// TwinCAT 3 PLC project AutoTune_PLC
// ProgramVersion: 3.1.4026.17
// libraries:
//   Tc2_MC2, * (Beckhoff Automation GmbH)
//   Tc2_Standard, * (Beckhoff Automation GmbH)
//   Tc2_System, * (Beckhoff Automation GmbH)
//   Tc3_Module, * (Beckhoff Automation GmbH)
//   VisuDialogs, * (System)
//   VisuSymbols,newest,System
// project tree:
//   / GlobalTextList.TcGTLO (not stored), PlcTask.TcTTO (not stored), Visualization Manager.TcVMO (not stored)
//   GVLs/ GVLSafeIO.TcGVL (not stored), GVLStdIO.TcGVL (not stored)
//   POUs/ FB_Blinker.TcPOU (not stored), MAIN.TcPOU
//   VISUs/ Visualization.TcVIS (not stored)
// real-time tasks:
//   TASK PlcTask: cycle T#10ms, priority 40, ADS port 350
// motion (NC):
//   TASK NC-Task 1 SAF: cycle T#2ms, priority 4, ADS port 501
//   TASK NC-Task 1 SVB: cycle T#10ms, priority 8, ADS port 511
//   AXIS Axis 1 (id 1)
//     General: UnitName=°
//     Dynamic: Acceleration=15000, Deceleration=15000, Jerk=69686.919
//     Velo: RefSearch=154.85982, RefSync=154.85982, SlowManual=774.2991, FastManual=4645.7946, Fast=15485.982, Maximum=15485.982
//     OtherSettings: AllowMotionCmdToSlave=true
//     encoder EncType=19
//       EncPara: ScaleFactorNumerator=360, ScaleFactorDenominator=1048576, MaxCount=#xffffffff
//     drive DrvType=16
//       DrvPara: MaxCount=#xffffffff, DriveControlDWord=#x00020100
//         Analog: VeloReferenz=17034.5802, VeloScale=71.5255737304688, TorqueSetpointScale=10, ScaleFactorActTorque=0.1
//         TimeComp: TaskDelayCycles=1
//     controller CtrType=1
//       CtrPara: PriorControlFactor=1
//         Observer: BandWidth=20
//   AXIS Axis 2 (id 2)
//     OtherSettings: AllowMotionCmdToSlave=true
//     encoder EncType=19
//       EncPara: MaxCount=#xffffffff
//     drive DrvType=16
//       DrvPara: MaxCount=#xffffffff, DriveControlDWord=#x00020100
//         Analog: TorqueSetpointScale=10, ScaleFactorActTorque=0.1
//         TimeComp: TaskDelayCycles=1
//     controller CtrType=1
//       CtrPara: PriorControlFactor=1
//         Observer: BandWidth=20
// I/O:
//   DEVICE Device 1 (EtherCAT), AmsNetId 5.143.164.192.2.1
//     Term 1 (EK1200) [EK1200-5000 EtherCAT Power supply (2A E-Bus)]
//       Term 2 (EL3214-0090) [EL3214-0090 4Ch. Ana. Input PT100 (RTD), TwinSAFE SC]
//       Term 3 (EL1904) [EL1904, 4 Ch. Safety Input 24V, TwinSAFE]
//         modules: Module 1 (FSOES)
//       Term 4 (EL2008) [EL2008 8Ch. Dig. Output 24V, 0.5A]
//       Term 5 (EL9011) [EL9011 End Terminal]
//   DEVICE Device 4 (EtherCAT), AmsNetId 5.143.164.192.5.1
//     Term 6 (AX8620-0000-0105) [AX8620-0000-0105]
//       Drive 7 (AX8206-0200-0106) [AX8206-0200-0106 (2Ch. 6A servo axis, safe-motion)]
//         modules: Device, Device, Device, Device, Device, Device, Device, Device, Device, Device, Device (Safety), Device, Device, Device, Device, Device, Device, Device, Device, Device, Device, Device, Device, Device, Device, Device, Device, Device, Device, Device, Device, Ch A, Ch A, Ch A, Ch A, Ch A, Ch A, Ch A, Ch A, Ch A, Ch A, Ch A, Ch A, Ch A, Ch A, Ch A, Ch A, Ch A, Ch A, Ch A, Ch A, Ch A, Ch A, Ch A, Ch A, Ch A, Ch A, Ch A, Ch A, Ch A, Ch A, Ch A, Ch B, Ch B, Ch B, Ch B, Ch B, Ch B, Ch B, Ch B, Ch B, Ch B, Ch B, Ch B, Ch B, Ch B, Ch B, Ch B, Ch B, Ch B, Ch B, Ch B, Ch B, Ch B, Ch B, Ch B, Ch B, Ch B
//         startup 12992:1 := 414D383034322D784A7830 // Ch A Motor parameters / Configured motor type
//         startup 24768:0 := FEFF // Ch A Interpolation sub mode select
//         startup 13000:5 := 0200 // Ch A Motor thermal model / Reaction
//         startup 13000:6 := 0000C841 // Ch A Motor thermal model / Partial fraction factor
//         startup 12992:12 := 0000FA45 // Ch A Motor parameters / Motor rated speed
//         startup 12992:13 := E6AE4540 // Ch A Motor parameters / Motor rated torque
//         startup 24694:0 := 03100000 // Ch A Motor standstill torque
//         startup 24800:0 := D007 // Ch A Positive torque/force limit value
//         startup 24801:0 := D007 // Ch A Negative torque/force limit value
//         startup 12288:6 := 4158383230362D303230302D30303030 // Ch A AxisMain parameters / Configured drive type
//         startup 12867:1 := CDCCDC40 // Ch A TorqueCtrl parameters / Configured channel rated current
//         startup 12867:2 := 0000A041 // Ch A TorqueCtrl parameters / Configured channel peak current
//         startup 12867:7 := 77BE1F40 // Ch A TorqueCtrl parameters / Iuvw max sum
//         startup 24672:0 := 08 // Ch A Modes of operation
//         startup 13023:0 := 0000 // Ch A Motor control mode
//         startup 12864:1 := 84C3B441 // Ch A TorqueCtrl parameters mappable / Torque control proportional gain q
//         startup 12864:2 := 8A0E7C39 // Ch A TorqueCtrl parameters mappable / Torque control integral action time q
//         startup 12608:1 := 9513BE3D // Ch A VeloCtrl parameters mappable / Velocity control proportional gain
//         startup 12608:2 := 6F12033C // Ch A VeloCtrl parameters mappable / Velocity control integral action time
//         startup 12608:3 := 00980546 // Ch A VeloCtrl parameters mappable / Bipolar velocity limit value
//         startup 12992:15 := 0100 // Ch A Motor parameters / Motor temperature sensor connection
//         startup 12611:4 := 0400 // Ch A VeloCtrl observer / Observer type
//         startup 24672:0 := 08 // Ch A Modes of operation
//         startup 12296:2 := 00 // Ch A AxisMain parameters encoder direction / Primary encoder direction
//   DEVICE Device 2 (EtherCAT Automation Protocol) (disabled), AmsNetId 5.143.164.192.3.1
//   DEVICE Device 3 (COM Port) (disabled)
//   DEVICE Device 7 (COM Port) (disabled)
// variable links:
//   Device 1 (EtherCAT) <-> Device 4 (EtherCAT)/Term 6 (AX8620-0000-0105)/Drive 7 (AX8206-0200-0106)
//     Term 1 (EK1200)/Term 3 (EL1904)/Module 1 (FSOES)/RxPDO/FSOE <-> Device (Safety)/FSoE Master Connection 1 Master Message/Message_3
//     Term 1 (EK1200)/Term 3 (EL1904)/Module 1 (FSOES)/TxPDO/FSOE <-> Device (Safety)/FSoE Master Connection 1 Slave Message/Message_3
//   Device 4 (EtherCAT) <-> Device 4 (EtherCAT)/Term 6 (AX8620-0000-0105)
//     Term 6 (AX8620-0000-0105)/Drive 7 (AX8206-0200-0106)/Device/DeviceMain Outputs/Power supply controlword <-> PSM Controlword for axis/Controlword for axis
//   NC-Task 1 SAF/Axes/Axis 1 <-> Device 4 (EtherCAT)/Term 6 (AX8620-0000-0105)/Drive 7 (AX8206-0200-0106)
//     Drive/Inputs/In/nDataIn1 <-> Ch A/Ch A PositionControl Inputs/Ch A Following error actual value
//     Drive/Inputs/In/nDataIn3[0] <-> Ch A/Ch A TorqueControl Inputs/Ch A Torque/force actual value
//     Drive/Inputs/In/nDcOutputTime <-> InfoData/DcOutputShift
//     Drive/Inputs/In/nState1 <-> Ch A/Ch A AxisMain Inputs/Ch A Statusword
//     Drive/Inputs/In/nState2 <-> Ch A/Ch A AxisMain Inputs/Ch A Statusword @bit 8
//     Drive/Inputs/In/nState4 @bit 1 <-> WcState/InputToggle0
//     Drive/Inputs/In/nState4 <-> WcState/WcState0
//     Drive/Outputs/Out/nCtrl1 <-> Ch A/Ch A AxisMain Outputs/Ch A Controlword
//     Drive/Outputs/Out/nCtrl2 <-> Ch A/Ch A AxisMain Outputs/Ch A Controlword @bit 8
//     Drive/Outputs/Out/nDataOut1 <-> Ch A/Ch A Interpolator Outputs/Ch A Target position
//     Drive/Outputs/Out/nDataOut2 <-> Ch A/Ch A Interpolator Outputs/Ch A Target velocity
//     Enc/Inputs/In/nDataIn1 <-> Ch A/Ch A AxisMain Inputs/Ch A Position actual value
//     Enc/Inputs/In/nDcInputTime <-> InfoData/DcInputShift
//     Enc/Inputs/In/nState2 @bit 5 <-> Ch A/Ch A AxisMain Inputs/Position actual value invalid
//     Enc/Inputs/In/nState4 @bit 1 <-> WcState/InputToggle0
//     Enc/Inputs/In/nState4 <-> WcState/WcState0
//   NC-Task 1 SAF/Axes/Axis 2 <-> Device 4 (EtherCAT)/Term 6 (AX8620-0000-0105)/Drive 7 (AX8206-0200-0106)
//     Drive/Inputs/In/nDataIn1 <-> Ch B/Ch B PositionControl Inputs/Ch B Following error actual value
//     Drive/Inputs/In/nDcOutputTime <-> InfoData/DcOutputShift
//     Drive/Inputs/In/nState1 <-> Ch B/Ch B AxisMain Inputs/Ch B Statusword
//     Drive/Inputs/In/nState2 <-> Ch B/Ch B AxisMain Inputs/Ch B Statusword @bit 8
//     Drive/Inputs/In/nState4 @bit 1 <-> WcState/InputToggle0
//     Drive/Inputs/In/nState4 <-> WcState/WcState0
//     Drive/Outputs/Out/nCtrl1 <-> Ch B/Ch B AxisMain Outputs/Ch B Controlword
//     Drive/Outputs/Out/nCtrl2 <-> Ch B/Ch B AxisMain Outputs/Ch B Controlword @bit 8
//     Drive/Outputs/Out/nDataOut1 <-> Ch B/Ch B Interpolator Outputs/Ch B Target position
//     Drive/Outputs/Out/nDataOut2 <-> Ch B/Ch B Interpolator Outputs/Ch B Target velocity
//     Enc/Inputs/In/nDataIn1 <-> Ch B/Ch B AxisMain Inputs/Ch B Position actual value
//     Enc/Inputs/In/nDcInputTime <-> InfoData/DcInputShift
//     Enc/Inputs/In/nState2 @bit 5 <-> Ch B/Ch B AxisMain Inputs/Position actual value invalid
//     Enc/Inputs/In/nState4 @bit 1 <-> WcState/InputToggle0
//     Enc/Inputs/In/nState4 <-> WcState/WcState0
//   AutoTune_PLC/AutoTune_PLC Instance <-> Device 1 (EtherCAT)/Term 1 (EK1200)/Term 2 (EL3214-0090)
//     PlcTask Inputs/GVLStdIO._PotInput <-> RTD Inputs Channel 1/Value
//   AutoTune_PLC/AutoTune_PLC Instance <-> Device 1 (EtherCAT)/Term 1 (EK1200)/Term 3 (EL1904)
//     PlcTask Inputs/GVLSafeIO._es1Status <-> Module 1 (FSOES)/TxPDO/FSOE/InputChannel1
//     PlcTask Inputs/GVLSafeIO._es2Status <-> Module 1 (FSOES)/TxPDO/FSOE/InputChannel2
//     PlcTask Inputs/GVLSafeIO._pbRestart <-> Module 1 (FSOES)/TxPDO/FSOE/InputChannel3
//   AutoTune_PLC/AutoTune_PLC Instance <-> Device 1 (EtherCAT)/Term 1 (EK1200)/Term 4 (EL2008)
//     PlcTask Outputs/GVLStdIO._ResetLt <-> Channel 1/Output
//   AutoTune_PLC/AutoTune_PLC Instance <-> Device 4 (EtherCAT)/Term 6 (AX8620-0000-0105)/Drive 7 (AX8206-0200-0106)
//     PlcTask Inputs/GVLSafeIO._TSG1_Comm_Err <-> Device (Safety)/Standard Inputdata/Standard Out Var 6
//     PlcTask Inputs/GVLSafeIO._TSG1_FB_Err <-> Device (Safety)/Standard Inputdata/Standard Out Var 5
//     PlcTask Inputs/GVLSafeIO._TSG1_Other_Err <-> Device (Safety)/Standard Inputdata/Standard Out Var 7
//     PlcTask Inputs/GVLSafeIO._TSG1_esOut <-> Device (Safety)/Standard Inputdata/Standard Out Var 11
//     PlcTask Inputs/GVLSafeIO._esError <-> Device (Safety)/Standard Inputdata/Standard Out Var 8
//     PlcTask Outputs/GVLSafeIO._TSG1_ErrAck <-> Device (Safety)/Standard Outputdata/Standard In Var 1
//     PlcTask Outputs/GVLSafeIO._TSG1_Run <-> Device (Safety)/Standard Outputdata/Standard In Var 2
//   AutoTune_PLC/AutoTune_PLC Instance <-> NC-Task 1 SAF/Axes/Axis 1
//     PlcTask Inputs/MAIN.A1.NcToPlc <-> Outputs/ToPlc
//     PlcTask Outputs/MAIN.A1.PlcToNc <-> Inputs/FromPlc

// ---- POUs/MAIN.TcPOU
PROGRAM MAIN
VAR
	_SpeedOverride : LREAL;
	FastBlink: FB_Blinker;
	SlowBlink: FB_Blinker;
	
	testtmr : TON;
	
	A1 : AXIS_REF;

	//Enable
	A1Pwr : MC_POWER;
	bA1Enable: BOOL;
	bA1PwrStatus: BOOL;
	bA1PwrBusy: BOOL;
	bA1PwrError: BOOL;
	bA1PwrErrorId: UDINT;
	
	bA1PwrErrorLatch: BOOL;
	
	//Reset
	A1Reset : MC_RESET;
	bA1Reset: BOOL;
	bA1ResetDone: BOOL;
	bA1ResetBusy: BOOL;
	bA1Error: BOOL;
	bA1ErrorId: UDINT;
	
	//Jog
	A1Jog : MC_JOG;
	bA1JogFwd: BOOL;
	bA1JogRev: BOOL;
	bA1JogMode: E_JogMode := MC_JOGMODE_CONTINOUS;
	bA1JogPosition: LREAL;
	bA1JogVelocity: LREAL := 1000;
	bA1JogAccel: LREAL := 5000;
	bA1JogDecel: LREAL := 5000;
	bA1JogJerk: LREAL := 10000;
	bA1JogDone: BOOL;
	bA1JogBusy: BOOL;
	bA1JogActive: BOOL;
	bA1JogCmdAborted: BOOL;
	bA1JogError: BOOL;
	bA1JogErrorId: UDINT;


	bA1PwrErrorIdLatch: UDINT;
	
	EnableDly : TON;
	
END_VAR

GVLSafeIO._TSG1_Run := TRUE;

GVLSafeIO._TSG1_ErrAck := GVLSafeIO._pbRestart;

//Make sure both contacts are in sync before pulsing light

//Controls Blink Of PB Lt

IF GVLSafeIO._TSG1_FB_Err OR GVLSafeIO._TSG1_Comm_Err OR GVLSafeIO._TSG1_Other_Err OR GVLSafeIO._esError THEN
	FastBlink(TmrPreset:= T#100MS, xOut=> GVLStdIO._ResetLt);
ELSIF NOT GVLSafeIO._TSG1_esOut AND GVLSafeIO._es1Status AND GVLSafeIO._es2Status THEN
	SlowBlink(TmrPreset:= T#1S, xOut=> GVLStdIO._ResetLt);
ELSIF NOT GVLSafeIO._es1Status OR NOT GVLSafeIO._es2Status THEN
	GVLStdIO._ResetLt := FALSE;
ELSIF GVLSafeIO._TSG1_esOut THEN
	GVLStdIO._ResetLt := TRUE;
END_IF

IF NOT bA1Enable THEN
	EnableDly(IN:= GVLSafeIO._pbRestart, PT:= T#2S, Q=> , ET=> );
		IF EnableDly.Q THEN
			bA1Enable := GVLSafeIO._pbRestart;
		END_IF
ELSIF NOT GVLSafeIO._TSG1_esOut THEN
			bA1Enable := FALSE;
END_IF

bA1Reset := GVLSafeIO._pbRestart;

//Scale POT to 0-100% for speed override.
Scale();

A1Pwr(
	Axis:= A1, 
	Enable:= bA1Enable, 
	Enable_Positive:= TRUE, 
	Enable_Negative:= TRUE, 
	Override:= _SpeedOverride, 
	Status=> bA1PwrStatus, 
	Busy=> bA1PwrBusy, 
	Error=> bA1PwrError, 
	ErrorID=> bA1PwrErrorId);
	
IF bA1PwrError THEN
	bA1PwrErrorLatch := TRUE;
	bA1PwrErrorIdLatch := bA1PwrErrorId; 
END_IF
	
IF bA1Reset THEN
	bA1PwrErrorLatch := FALSE;
	bA1PwrErrorIdLatch := 0; 
END_IF



A1Reset(
	Axis:= A1, 
	Execute:= bA1Reset, 
	Done=> bA1ResetDone, 
	Busy=> bA1ResetBusy, 
	Error=> bA1Error, 
	ErrorID=> bA1ErrorId);

A1Jog(
	Axis:= A1, 
	JogForward:= bA1JogFwd, 
	JogBackwards:= bA1JogRev, 
	Mode:= bA1JogMode, 
	Position:= bA1JogPosition, 
	Velocity:= bA1JogVelocity, 
	Acceleration:= bA1JogAccel, 
	Deceleration:= bA1JogDecel, 
	Jerk:= bA1JogJerk, 
	Done=> bA1JogDone, 
	Busy=> bA1JogBusy, 
	Active=> bA1JogActive, 
	CommandAborted=> bA1JogCmdAborted, 
	Error=> bA1JogError, 
	ErrorID=> bA1JogErrorId);
	
IF bA1Reset THEN
	bA1Reset := FALSE;
END_IF

ACTION Scale:
_SpeedOverride := (100.0 / 32767.0)*GVLStdIO._PotInput;
END_ACTION

END_PROGRAM
